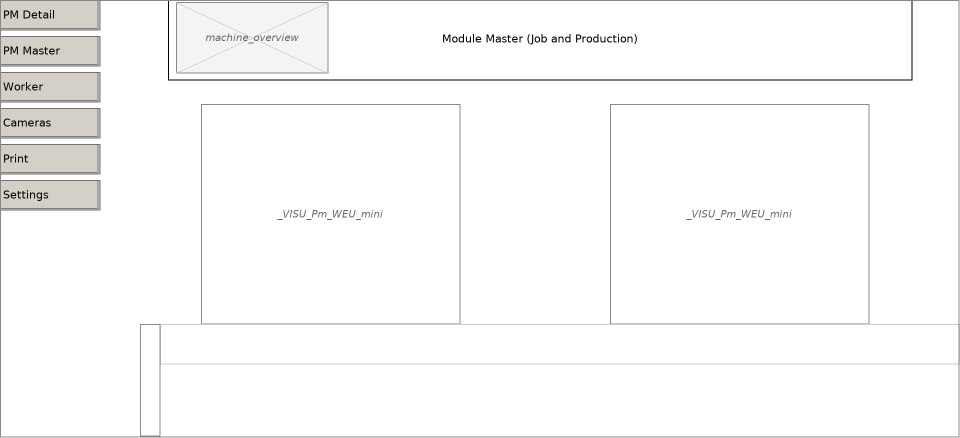
VISUALIZATION VISU_PrintOverview  // 960x438
    Button (0,144 100x30), "Print"
        OnMouseClick: change screen: VISU_PRINT
    Button (0,0 100x30), "PM Detail"
        OnMouseClick: change screen: VISU_PrintModule_Detail
    Button (0,72 100x30), "Worker"
        OnMouseClick: change screen: VISU_Workers
    Frame (610,104 259x220)
        shows _VISU_Pm_WEU_mini(mInst := PRG_PRINT.fbPrintModule[1])
    Frame (201,104 259x220)
        shows _VISU_Pm_WEU_mini(mInst := PRG_PRINT.fbPrintModule[2])
    Rectangle (160,324 800x40), colour toggle: PRG_PRINT.fbPrintOverview.bMovingInd
    Frame (140,324 20x112)
        shows CalmarProdDmax._VISU_CTsFlow(m_Inst := PRG_PRINT.fbPrintOverview)
    RoundedRectangle (168,-2 744x82), "Module Master (Job and Production)"
    Image (176,2 152x71), image: machine_overview
    Button (0,180 100x30), "Settings", input disabled if: TRUE
        OnMouseClick: change screen: VISU_SettingsWeu
    Button (0,108 100x30), "Cameras"
        OnMouseClick: change screen: VISU_Cameras
    Button (0,36 100x30), "PM Master", input disabled if: TRUE
        OnMouseClick: change screen: VISU_ModuleMaster
END_VISUALIZATION

(* stored: Version 1.1.0.1, ProductVersion 3.1.4024.11
   Visu VISU_PrintOverview: Id {a6ed15b6-9f2e-485d-8015-919bd40398e8} *)
